{attribute 'GeneratedUsingTerminal: EM7004-0000-9996'}
{attribute addProperty BoxType "EM7004-0000-9996"}
{attribute addProperty Id "InputAT %I*ARRAY[0..15] OF BOOL16"}
{attribute addProperty CRC "2621435360"}
{attribute addProperty Size "16"}
TYPE DI_Inputs_BD004D6F EXTENDS InputBase_8311D824 :
STRUCT
	{attribute addProperty Name "Input"}
	Input AT %I* : ARRAY[0..15] OF BOOL;
END_STRUCT
END_TYPE

(* stored: Version 1.2.0.0, ProductVersion 3.1.4024.11
   DUT DI_Inputs_BD004D6F: Id {ff67b166-bb16-437f-bcd7-00ef6320b8a7} *)
